// TIA Portal V19 export
DATA_BLOCK "Alarmtimer"   // DB26
{ S7_Optimized_Access := 'TRUE' }
AUTHOR : FLA
FAMILY : UHT
VERSION : 1.0
// stored: AutoNumber false, MemoryReserve 0
   VAR RETAIN
      System : Word;   // System
      DBW2 : Word;
      DBW4 : Word;
      DBW6 : Word;
      DBW8 : Word;
      DBW10 : Word;
   END_VAR
BEGIN
END_DATA_BLOCK
